// TIA Portal V17 export
// export: Created 2022-05-07T16:38:47.6768571Z, ExportSetting WithDefaults, DisplayName Totally Integrated Automation Portal, DisplayVersion V17 Update 3, DisplayName TIA Portal Openness, DisplayVersion V17 Update 3, DisplayName TIA Portal Version Control Interface, DisplayVersion V17, DisplayName TIA Portal Test Suite Advanced, DisplayVersion V17 Update 1, DisplayName SINAMICS Startdrive Advanced, DisplayVersion V17 Update2, DisplayName SINAMICS Startdrive G130, G150, S120, S150, SINAMICS MV, S210, DisplayVersion V17 Update2, DisplayName SINAMICS Startdrive G110M, G120, G120C, G120D, G120P, G115D, DisplayVersion V17 Update2, DisplayName STEP 7 Professional, DisplayVersion V17 Update 3, DisplayName STEP 7 Safety, DisplayVersion V17, DisplayName WinCC UA Professional, DisplayVersion V17 Update 3
FUNCTION_BLOCK "FB_ORG_ASSI"   // FB5, LAD
{ S7_Optimized_Access := 'TRUE' }
VERSION : 0.1
// stored: AutoNumber true, IsIECCheckEnabled false, IsRetainMemResEnabled false, MemoryReserve 100, SetENOAutomatically false, UDAEnableTagReadback false
   VAR
      CTRL_ASSE_STD_MA { S7_SetPoint := 'True'} : "CTRL_ASSE_STD";
      CTRL_ASSE_STD_MR { S7_SetPoint := 'True'} : "CTRL_ASSE_STD";
      CTRL_ASSE_STD_MS { S7_SetPoint := 'True'} : "CTRL_ASSE_STD";
      CTRL_ASSE_STD_ME { S7_SetPoint := 'True'} : "CTRL_ASSE_STD";
   END_VAR
BEGIN

REGION Network 1: RESET ALLARMI
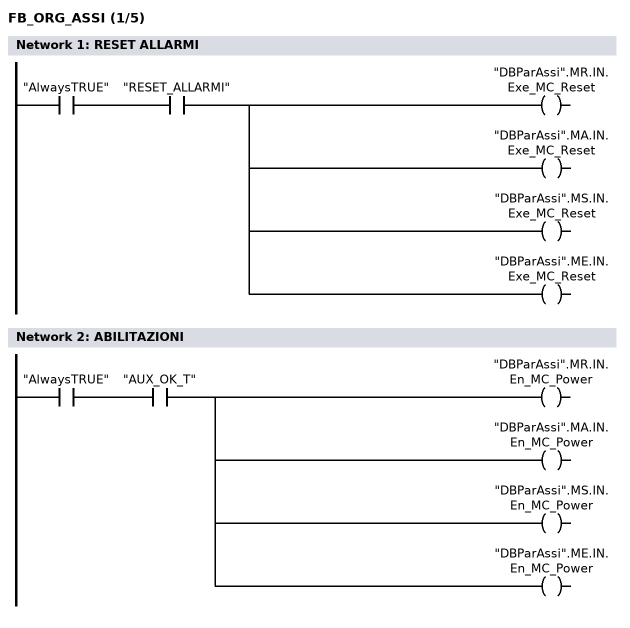
   RUNG wire#powerrail
      Contact( "AlwaysTRUE" )
      Contact( "RESET_ALLARMI" )
      wire#w1
      Coil( "DBParAssi".MR.IN.Exe_MC_Reset )
   END_RUNG
   RUNG wire#w1
      Coil( "DBParAssi".MA.IN.Exe_MC_Reset )
   END_RUNG
   RUNG wire#w1
      Coil( "DBParAssi".MS.IN.Exe_MC_Reset )
   END_RUNG
   RUNG wire#w1
      Coil( "DBParAssi".ME.IN.Exe_MC_Reset )
   END_RUNG
   // the same network as SCL:
   "DBParAssi".MR.IN.Exe_MC_Reset := "AlwaysTRUE" AND "RESET_ALLARMI";
   "DBParAssi".MA.IN.Exe_MC_Reset := "DBParAssi".MR.IN.Exe_MC_Reset;
   "DBParAssi".MS.IN.Exe_MC_Reset := "DBParAssi".MR.IN.Exe_MC_Reset;
   "DBParAssi".ME.IN.Exe_MC_Reset := "DBParAssi".MR.IN.Exe_MC_Reset;
END_REGION

REGION Network 2: ABILITAZIONI
   RUNG wire#powerrail
      Contact( "AlwaysTRUE" )
      Contact( "AUX_OK_T" )
      wire#w1
      Coil( "DBParAssi".MR.IN.En_MC_Power )
   END_RUNG
   RUNG wire#w1
      Coil( "DBParAssi".MA.IN.En_MC_Power )
   END_RUNG
   RUNG wire#w1
      Coil( "DBParAssi".MS.IN.En_MC_Power )
   END_RUNG
   RUNG wire#w1
      Coil( "DBParAssi".ME.IN.En_MC_Power )
   END_RUNG
   // the same network as SCL:
   "DBParAssi".MR.IN.En_MC_Power := "AlwaysTRUE" AND "AUX_OK_T";
   "DBParAssi".MA.IN.En_MC_Power := "DBParAssi".MR.IN.En_MC_Power;
   "DBParAssi".MS.IN.En_MC_Power := "DBParAssi".MR.IN.En_MC_Power;
   "DBParAssi".ME.IN.En_MC_Power := "DBParAssi".MR.IN.En_MC_Power;
END_REGION

REGION Network 3: ISTANZA MR
   // homing attivo = 3
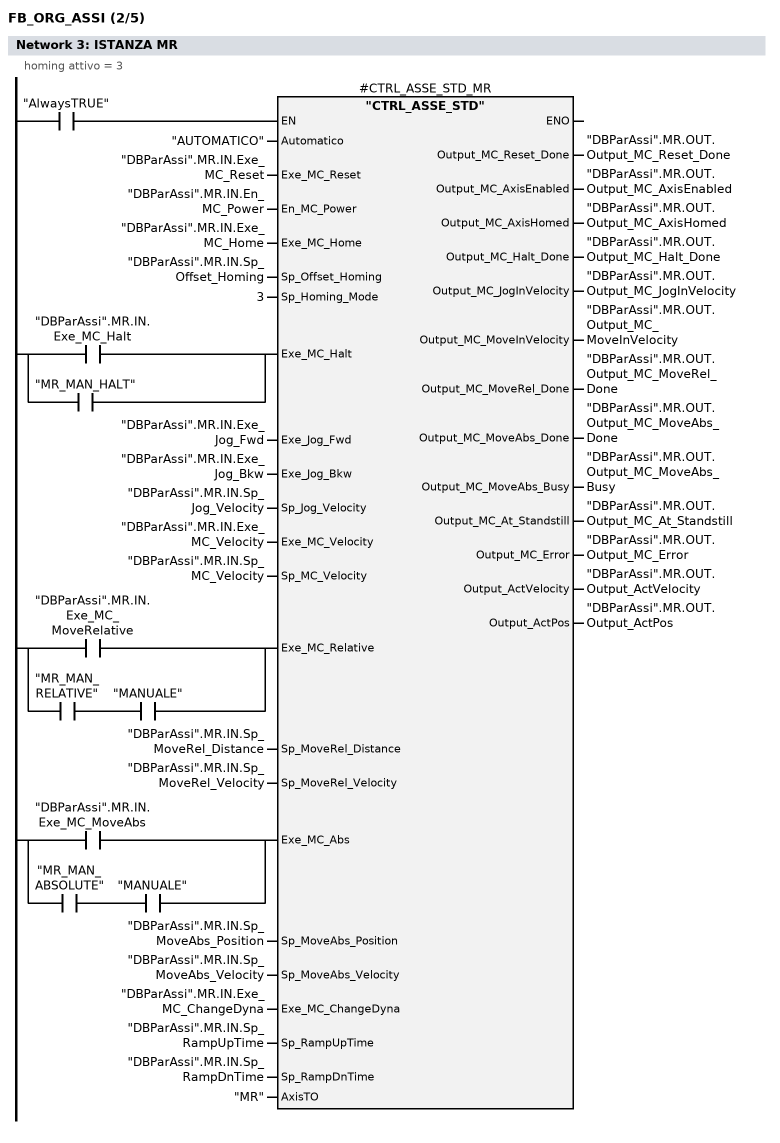
   RUNG wire#powerrail
      Contact( "AlwaysTRUE" )
      #CTRL_ASSE_STD_MR(Exe_MC_Halt := wire#w1, Exe_MC_Relative := wire#w2, Exe_MC_Abs := wire#w3, Automatico := "AUTOMATICO", Exe_MC_Reset := "DBParAssi".MR.IN.Exe_MC_Reset, En_MC_Power := "DBParAssi".MR.IN.En_MC_Power, Exe_MC_Home := "DBParAssi".MR.IN.Exe_MC_Home, Sp_Offset_Homing := "DBParAssi".MR.IN.Sp_Offset_Homing, Sp_Homing_Mode := 3, Exe_Jog_Fwd := "DBParAssi".MR.IN.Exe_Jog_Fwd, Exe_Jog_Bkw := "DBParAssi".MR.IN.Exe_Jog_Bkw, Sp_Jog_Velocity := "DBParAssi".MR.IN.Sp_Jog_Velocity, Exe_MC_Velocity := "DBParAssi".MR.IN.Exe_MC_Velocity, Sp_MC_Velocity := "DBParAssi".MR.IN.Sp_MC_Velocity, Sp_MoveRel_Distance := "DBParAssi".MR.IN.Sp_MoveRel_Distance, Sp_MoveRel_Velocity := "DBParAssi".MR.IN.Sp_MoveRel_Velocity, Sp_MoveAbs_Position := "DBParAssi".MR.IN.Sp_MoveAbs_Position, Sp_MoveAbs_Velocity := "DBParAssi".MR.IN.Sp_MoveAbs_Velocity, Exe_MC_ChangeDyna := "DBParAssi".MR.IN.Exe_MC_ChangeDyna, Sp_RampUpTime := "DBParAssi".MR.IN.Sp_RampUpTime, Sp_RampDnTime := "DBParAssi".MR.IN.Sp_RampDnTime, AxisTO := "MR", Output_MC_Reset_Done => "DBParAssi".MR.OUT.Output_MC_Reset_Done, Output_MC_AxisEnabled => "DBParAssi".MR.OUT.Output_MC_AxisEnabled, Output_MC_AxisHomed => "DBParAssi".MR.OUT.Output_MC_AxisHomed, Output_MC_Halt_Done => "DBParAssi".MR.OUT.Output_MC_Halt_Done, Output_MC_JogInVelocity => "DBParAssi".MR.OUT.Output_MC_JogInVelocity, Output_MC_MoveInVelocity => "DBParAssi".MR.OUT.Output_MC_MoveInVelocity, Output_MC_MoveRel_Done => "DBParAssi".MR.OUT.Output_MC_MoveRel_Done, Output_MC_MoveAbs_Done => "DBParAssi".MR.OUT.Output_MC_MoveAbs_Done, Output_MC_MoveAbs_Busy => "DBParAssi".MR.OUT.Output_MC_MoveAbs_Busy, Output_MC_At_Standstill => "DBParAssi".MR.OUT.Output_MC_At_Standstill, Output_MC_Error => "DBParAssi".MR.OUT.Output_MC_Error, Output_ActVelocity => "DBParAssi".MR.OUT.Output_ActVelocity, Output_ActPos => "DBParAssi".MR.OUT.Output_ActPos)
   END_RUNG
   RUNG wire#powerrail
      Contact( "DBParAssi".MR.IN.Exe_MC_Halt )
   END_RUNG wire#w1
   RUNG wire#powerrail
      Contact( "MR_MAN_HALT" )
   END_RUNG wire#w1
   RUNG wire#powerrail
      Contact( "DBParAssi".MR.IN.Exe_MC_MoveRelative )
   END_RUNG wire#w2
   RUNG wire#powerrail
      Contact( "MR_MAN_RELATIVE" )
      Contact( "MANUALE" )
   END_RUNG wire#w2
   RUNG wire#powerrail
      Contact( "DBParAssi".MR.IN.Exe_MC_MoveAbs )
   END_RUNG wire#w3
   RUNG wire#powerrail
      Contact( "MR_MAN_ABSOLUTE" )
      Contact( "MANUALE" )
   END_RUNG wire#w3
   // the same network as SCL:
   IF "AlwaysTRUE" THEN
       #CTRL_ASSE_STD_MR(Automatico := "AUTOMATICO",   // "CTRL_ASSE_STD"
                         Exe_MC_Reset := "DBParAssi".MR.IN.Exe_MC_Reset,
                         En_MC_Power := "DBParAssi".MR.IN.En_MC_Power,
                         Exe_MC_Home := "DBParAssi".MR.IN.Exe_MC_Home,
                         Sp_Offset_Homing := "DBParAssi".MR.IN.Sp_Offset_Homing,
                         Sp_Homing_Mode := 3,
                         Exe_MC_Halt := "DBParAssi".MR.IN.Exe_MC_Halt OR "MR_MAN_HALT",
                         Exe_Jog_Fwd := "DBParAssi".MR.IN.Exe_Jog_Fwd,
                         Exe_Jog_Bkw := "DBParAssi".MR.IN.Exe_Jog_Bkw,
                         Sp_Jog_Velocity := "DBParAssi".MR.IN.Sp_Jog_Velocity,
                         Exe_MC_Velocity := "DBParAssi".MR.IN.Exe_MC_Velocity,
                         Sp_MC_Velocity := "DBParAssi".MR.IN.Sp_MC_Velocity,
                         Exe_MC_Relative := "DBParAssi".MR.IN.Exe_MC_MoveRelative OR ("MR_MAN_RELATIVE" AND "MANUALE"),
                         Sp_MoveRel_Distance := "DBParAssi".MR.IN.Sp_MoveRel_Distance,
                         Sp_MoveRel_Velocity := "DBParAssi".MR.IN.Sp_MoveRel_Velocity,
                         Exe_MC_Abs := "DBParAssi".MR.IN.Exe_MC_MoveAbs OR ("MR_MAN_ABSOLUTE" AND "MANUALE"),
                         Sp_MoveAbs_Position := "DBParAssi".MR.IN.Sp_MoveAbs_Position,
                         Sp_MoveAbs_Velocity := "DBParAssi".MR.IN.Sp_MoveAbs_Velocity,
                         Exe_MC_ChangeDyna := "DBParAssi".MR.IN.Exe_MC_ChangeDyna,
                         Sp_RampUpTime := "DBParAssi".MR.IN.Sp_RampUpTime,
                         Sp_RampDnTime := "DBParAssi".MR.IN.Sp_RampDnTime,
                         AxisTO := "MR",
                         Output_MC_Reset_Done => "DBParAssi".MR.OUT.Output_MC_Reset_Done,
                         Output_MC_AxisEnabled => "DBParAssi".MR.OUT.Output_MC_AxisEnabled,
                         Output_MC_AxisHomed => "DBParAssi".MR.OUT.Output_MC_AxisHomed,
                         Output_MC_Halt_Done => "DBParAssi".MR.OUT.Output_MC_Halt_Done,
                         Output_MC_JogInVelocity => "DBParAssi".MR.OUT.Output_MC_JogInVelocity,
                         Output_MC_MoveInVelocity => "DBParAssi".MR.OUT.Output_MC_MoveInVelocity,
                         Output_MC_MoveRel_Done => "DBParAssi".MR.OUT.Output_MC_MoveRel_Done,
                         Output_MC_MoveAbs_Done => "DBParAssi".MR.OUT.Output_MC_MoveAbs_Done,
                         Output_MC_MoveAbs_Busy => "DBParAssi".MR.OUT.Output_MC_MoveAbs_Busy,
                         Output_MC_At_Standstill => "DBParAssi".MR.OUT.Output_MC_At_Standstill,
                         Output_MC_Error => "DBParAssi".MR.OUT.Output_MC_Error,
                         Output_ActVelocity => "DBParAssi".MR.OUT.Output_ActVelocity,
                         Output_ActPos => "DBParAssi".MR.OUT.Output_ActPos);
   END_IF;
END_REGION

REGION Network 4: ISTANZA MA
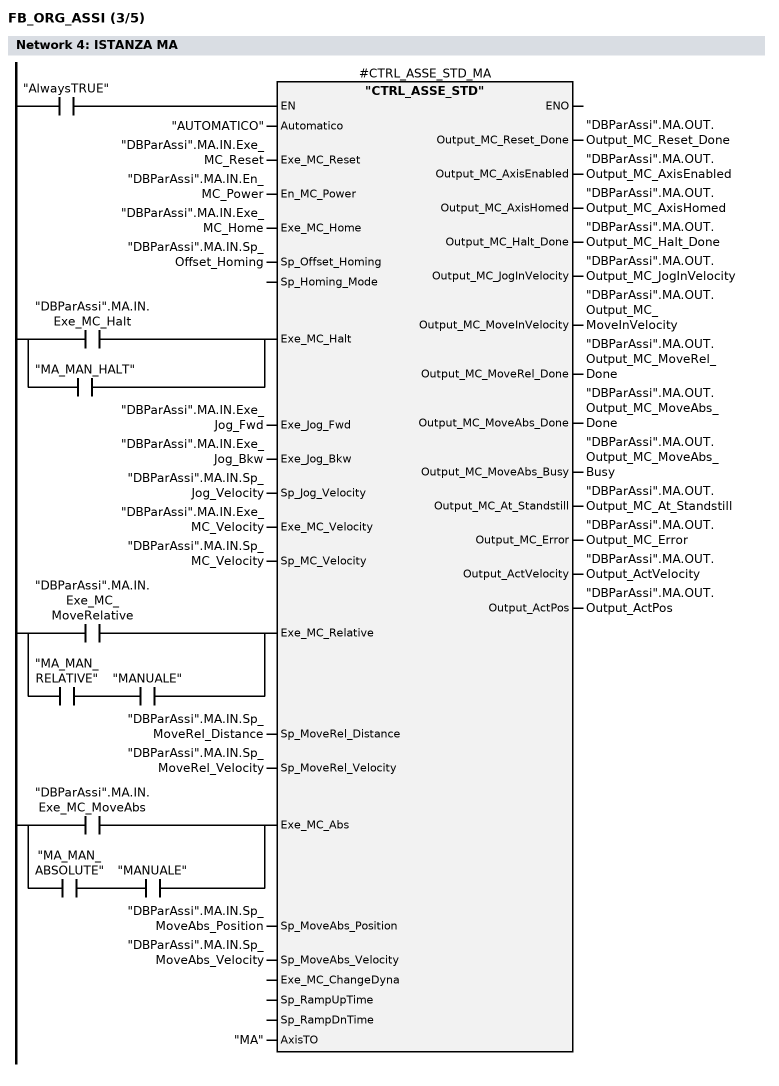
   RUNG wire#powerrail
      Contact( "AlwaysTRUE" )
      #CTRL_ASSE_STD_MA(Exe_MC_Halt := wire#w1, Exe_MC_Relative := wire#w2, Exe_MC_Abs := wire#w3, Automatico := "AUTOMATICO", Exe_MC_Reset := "DBParAssi".MA.IN.Exe_MC_Reset, En_MC_Power := "DBParAssi".MA.IN.En_MC_Power, Exe_MC_Home := "DBParAssi".MA.IN.Exe_MC_Home, Sp_Offset_Homing := "DBParAssi".MA.IN.Sp_Offset_Homing, Sp_Homing_Mode :=, Exe_Jog_Fwd := "DBParAssi".MA.IN.Exe_Jog_Fwd, Exe_Jog_Bkw := "DBParAssi".MA.IN.Exe_Jog_Bkw, Sp_Jog_Velocity := "DBParAssi".MA.IN.Sp_Jog_Velocity, Exe_MC_Velocity := "DBParAssi".MA.IN.Exe_MC_Velocity, Sp_MC_Velocity := "DBParAssi".MA.IN.Sp_MC_Velocity, Sp_MoveRel_Distance := "DBParAssi".MA.IN.Sp_MoveRel_Distance, Sp_MoveRel_Velocity := "DBParAssi".MA.IN.Sp_MoveRel_Velocity, Sp_MoveAbs_Position := "DBParAssi".MA.IN.Sp_MoveAbs_Position, Sp_MoveAbs_Velocity := "DBParAssi".MA.IN.Sp_MoveAbs_Velocity, Exe_MC_ChangeDyna :=, Sp_RampUpTime :=, Sp_RampDnTime :=, AxisTO := "MA", Output_MC_Reset_Done => "DBParAssi".MA.OUT.Output_MC_Reset_Done, Output_MC_AxisEnabled => "DBParAssi".MA.OUT.Output_MC_AxisEnabled, Output_MC_AxisHomed => "DBParAssi".MA.OUT.Output_MC_AxisHomed, Output_MC_Halt_Done => "DBParAssi".MA.OUT.Output_MC_Halt_Done, Output_MC_JogInVelocity => "DBParAssi".MA.OUT.Output_MC_JogInVelocity, Output_MC_MoveInVelocity => "DBParAssi".MA.OUT.Output_MC_MoveInVelocity, Output_MC_MoveRel_Done => "DBParAssi".MA.OUT.Output_MC_MoveRel_Done, Output_MC_MoveAbs_Done => "DBParAssi".MA.OUT.Output_MC_MoveAbs_Done, Output_MC_MoveAbs_Busy => "DBParAssi".MA.OUT.Output_MC_MoveAbs_Busy, Output_MC_At_Standstill => "DBParAssi".MA.OUT.Output_MC_At_Standstill, Output_MC_Error => "DBParAssi".MA.OUT.Output_MC_Error, Output_ActVelocity => "DBParAssi".MA.OUT.Output_ActVelocity, Output_ActPos => "DBParAssi".MA.OUT.Output_ActPos)
   END_RUNG
   RUNG wire#powerrail
      Contact( "DBParAssi".MA.IN.Exe_MC_Halt )
   END_RUNG wire#w1
   RUNG wire#powerrail
      Contact( "MA_MAN_HALT" )
   END_RUNG wire#w1
   RUNG wire#powerrail
      Contact( "DBParAssi".MA.IN.Exe_MC_MoveRelative )
   END_RUNG wire#w2
   RUNG wire#powerrail
      Contact( "MA_MAN_RELATIVE" )
      Contact( "MANUALE" )
   END_RUNG wire#w2
   RUNG wire#powerrail
      Contact( "DBParAssi".MA.IN.Exe_MC_MoveAbs )
   END_RUNG wire#w3
   RUNG wire#powerrail
      Contact( "MA_MAN_ABSOLUTE" )
      Contact( "MANUALE" )
   END_RUNG wire#w3
   // the same network as SCL:
   IF "AlwaysTRUE" THEN
       #CTRL_ASSE_STD_MA(Automatico := "AUTOMATICO",   // "CTRL_ASSE_STD"
                         Exe_MC_Reset := "DBParAssi".MA.IN.Exe_MC_Reset,
                         En_MC_Power := "DBParAssi".MA.IN.En_MC_Power,
                         Exe_MC_Home := "DBParAssi".MA.IN.Exe_MC_Home,
                         Sp_Offset_Homing := "DBParAssi".MA.IN.Sp_Offset_Homing,
                         Exe_MC_Halt := "DBParAssi".MA.IN.Exe_MC_Halt OR "MA_MAN_HALT",
                         Exe_Jog_Fwd := "DBParAssi".MA.IN.Exe_Jog_Fwd,
                         Exe_Jog_Bkw := "DBParAssi".MA.IN.Exe_Jog_Bkw,
                         Sp_Jog_Velocity := "DBParAssi".MA.IN.Sp_Jog_Velocity,
                         Exe_MC_Velocity := "DBParAssi".MA.IN.Exe_MC_Velocity,
                         Sp_MC_Velocity := "DBParAssi".MA.IN.Sp_MC_Velocity,
                         Exe_MC_Relative := "DBParAssi".MA.IN.Exe_MC_MoveRelative OR ("MA_MAN_RELATIVE" AND "MANUALE"),
                         Sp_MoveRel_Distance := "DBParAssi".MA.IN.Sp_MoveRel_Distance,
                         Sp_MoveRel_Velocity := "DBParAssi".MA.IN.Sp_MoveRel_Velocity,
                         Exe_MC_Abs := "DBParAssi".MA.IN.Exe_MC_MoveAbs OR ("MA_MAN_ABSOLUTE" AND "MANUALE"),
                         Sp_MoveAbs_Position := "DBParAssi".MA.IN.Sp_MoveAbs_Position,
                         Sp_MoveAbs_Velocity := "DBParAssi".MA.IN.Sp_MoveAbs_Velocity,
                         AxisTO := "MA",
                         Output_MC_Reset_Done => "DBParAssi".MA.OUT.Output_MC_Reset_Done,
                         Output_MC_AxisEnabled => "DBParAssi".MA.OUT.Output_MC_AxisEnabled,
                         Output_MC_AxisHomed => "DBParAssi".MA.OUT.Output_MC_AxisHomed,
                         Output_MC_Halt_Done => "DBParAssi".MA.OUT.Output_MC_Halt_Done,
                         Output_MC_JogInVelocity => "DBParAssi".MA.OUT.Output_MC_JogInVelocity,
                         Output_MC_MoveInVelocity => "DBParAssi".MA.OUT.Output_MC_MoveInVelocity,
                         Output_MC_MoveRel_Done => "DBParAssi".MA.OUT.Output_MC_MoveRel_Done,
                         Output_MC_MoveAbs_Done => "DBParAssi".MA.OUT.Output_MC_MoveAbs_Done,
                         Output_MC_MoveAbs_Busy => "DBParAssi".MA.OUT.Output_MC_MoveAbs_Busy,
                         Output_MC_At_Standstill => "DBParAssi".MA.OUT.Output_MC_At_Standstill,
                         Output_MC_Error => "DBParAssi".MA.OUT.Output_MC_Error,
                         Output_ActVelocity => "DBParAssi".MA.OUT.Output_ActVelocity,
                         Output_ActPos => "DBParAssi".MA.OUT.Output_ActPos);
   END_IF;
END_REGION

REGION Network 5 (SCL): ISTANZA MA SCL

   // #CTRL_ASSE_STD_MA(Exe_MC_Reset:="DBParAssi".MA.IN.Exe_MC_Reset,
   //                         En_MC_Power:="DBParAssi".MA.IN.En_MC_Power,
   //                         Exe_MC_Home:="DBParAssi".MA.IN.Exe_MC_Home,
   //                         Sp_Offset_Homing:="DBParAssi".MA.IN.Sp_Offset_Homing,
   //                         Exe_MC_Halt:="DBParAssi".MA.IN.Exe_MC_Halt,
   //                         Exe_Jog_Fwd:="DBParAssi".MA.IN.Exe_Jog_Fwd,
   //                         Exe_Jog_Bkw:="DBParAssi".MA.IN.Exe_Jog_Bkw,
   //                         Sp_Jog_Velocity:="DBParAssi".MA.IN.Sp_Jog_Velocity,
   //                         Exe_MC_Velocity:="DBParAssi".MA.IN.Exe_MC_Velocity,
   //                         Sp_MC_Velocity:="DBParAssi".MA.IN.Sp_MC_Velocity,
   //                         Exe_MC_Relative:="DBParAssi".MA.IN.Exe_MC_MoveRelative,
   //                         Sp_MoveRel_Distance:="DBParAssi".MA.IN.Sp_MoveRel_Distance,
   //                         Sp_MoveRel_Velocity:="DBParAssi".MA.IN.Sp_MoveRel_Velocity,
   //                         Exe_MC_Abs:="DBParAssi".MA.IN.Exe_MC_MoveAbs,
   //                         Sp_MoveAbs_Position:="DBParAssi".MA.IN.Sp_MoveAbs_Position,
   //                         Sp_MoveAbs_Velocity:="DBParAssi".MA.IN.Sp_MoveAbs_Velocity,
   //                         Output_MC_Reset_Done=>"DBParAssi".MA.OUT.Output_MC_Reset_Done,
   //                         Output_MC_AxisEnabled=>"DBParAssi".MA.OUT.Output_MC_AxisEnabled,
   //                         Output_MC_AxisHomed=>"DBParAssi".MA.OUT.Output_MC_AxisHomed,
   //                         Output_MC_Halt_Done=>"DBParAssi".MA.OUT.Output_MC_Halt_Done,
   //                         Output_MC_JogInVelocity=>"DBParAssi".MA.OUT.Output_MC_Reset_Done,
   //                         Output_MC_MoveInVelocity=>"DBParAssi".MA.OUT.Output_MC_MoveInVelocity,
   //                         Output_MC_MoveRel_Done=>"DBParAssi".MA.OUT.Output_MC_MoveRel_Done,
   //                         Output_MC_MoveAbs_Done=>"DBParAssi".MA.OUT.Output_MC_MoveAbs_Done,
   //                         Output_MC_MoveAbs_Busy=>"DBParAssi".MA.OUT.Output_MC_MoveAbs_Busy,
   //                         Output_MC_At_Standstill=>"DBParAssi".MA.OUT.Output_MC_Reset_Done,
   //                         Output_MC_Error=>"DBParAssi".MA.OUT.Output_MC_Error,
   //                         Output_ActVelocity=>"DBParAssi".MA.OUT.Output_ActVelocity,
   //                         Output_ActPos=>"DBParAssi".MA.OUT.Output_ActPos,
   //                         AxisTO:="MA");
END_REGION

REGION Network 6: ISTANZA MS
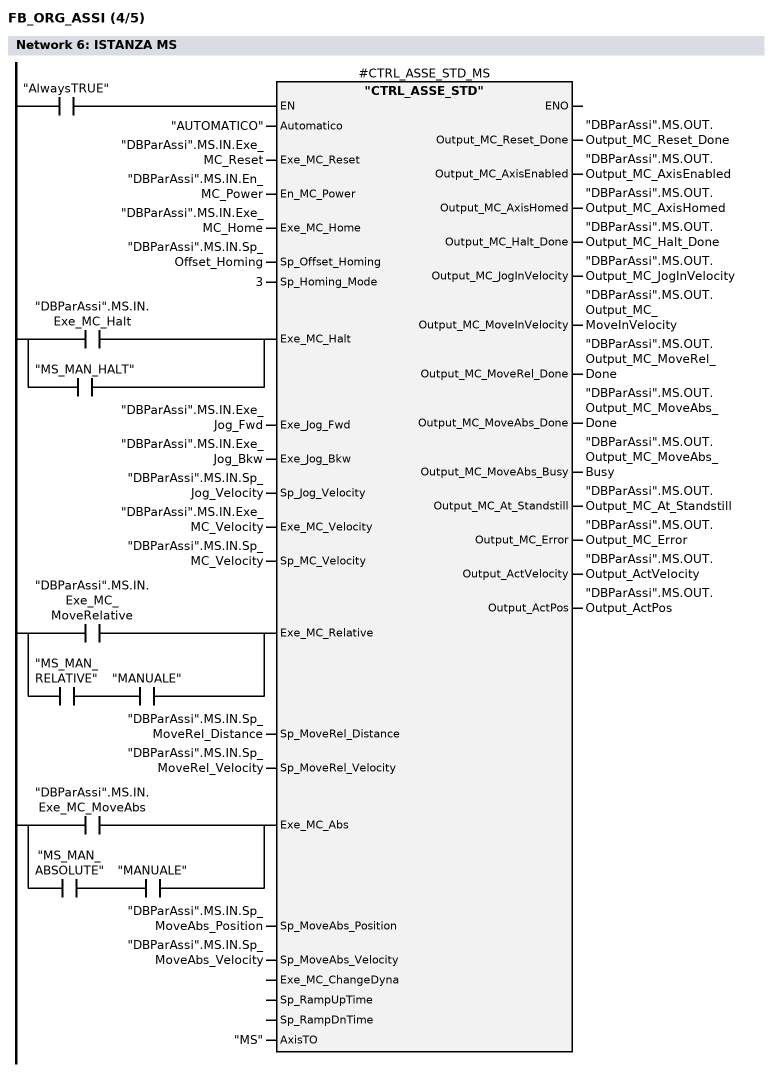
   RUNG wire#powerrail
      Contact( "AlwaysTRUE" )
      #CTRL_ASSE_STD_MS(Exe_MC_Halt := wire#w1, Exe_MC_Relative := wire#w2, Exe_MC_Abs := wire#w3, Automatico := "AUTOMATICO", Exe_MC_Reset := "DBParAssi".MS.IN.Exe_MC_Reset, En_MC_Power := "DBParAssi".MS.IN.En_MC_Power, Exe_MC_Home := "DBParAssi".MS.IN.Exe_MC_Home, Sp_Offset_Homing := "DBParAssi".MS.IN.Sp_Offset_Homing, Sp_Homing_Mode := 3, Exe_Jog_Fwd := "DBParAssi".MS.IN.Exe_Jog_Fwd, Exe_Jog_Bkw := "DBParAssi".MS.IN.Exe_Jog_Bkw, Sp_Jog_Velocity := "DBParAssi".MS.IN.Sp_Jog_Velocity, Exe_MC_Velocity := "DBParAssi".MS.IN.Exe_MC_Velocity, Sp_MC_Velocity := "DBParAssi".MS.IN.Sp_MC_Velocity, Sp_MoveRel_Distance := "DBParAssi".MS.IN.Sp_MoveRel_Distance, Sp_MoveRel_Velocity := "DBParAssi".MS.IN.Sp_MoveRel_Velocity, Sp_MoveAbs_Position := "DBParAssi".MS.IN.Sp_MoveAbs_Position, Sp_MoveAbs_Velocity := "DBParAssi".MS.IN.Sp_MoveAbs_Velocity, Exe_MC_ChangeDyna :=, Sp_RampUpTime :=, Sp_RampDnTime :=, AxisTO := "MS", Output_MC_Reset_Done => "DBParAssi".MS.OUT.Output_MC_Reset_Done, Output_MC_AxisEnabled => "DBParAssi".MS.OUT.Output_MC_AxisEnabled, Output_MC_AxisHomed => "DBParAssi".MS.OUT.Output_MC_AxisHomed, Output_MC_Halt_Done => "DBParAssi".MS.OUT.Output_MC_Halt_Done, Output_MC_JogInVelocity => "DBParAssi".MS.OUT.Output_MC_JogInVelocity, Output_MC_MoveInVelocity => "DBParAssi".MS.OUT.Output_MC_MoveInVelocity, Output_MC_MoveRel_Done => "DBParAssi".MS.OUT.Output_MC_MoveRel_Done, Output_MC_MoveAbs_Done => "DBParAssi".MS.OUT.Output_MC_MoveAbs_Done, Output_MC_MoveAbs_Busy => "DBParAssi".MS.OUT.Output_MC_MoveAbs_Busy, Output_MC_At_Standstill => "DBParAssi".MS.OUT.Output_MC_At_Standstill, Output_MC_Error => "DBParAssi".MS.OUT.Output_MC_Error, Output_ActVelocity => "DBParAssi".MS.OUT.Output_ActVelocity, Output_ActPos => "DBParAssi".MS.OUT.Output_ActPos)
   END_RUNG
   RUNG wire#powerrail
      Contact( "DBParAssi".MS.IN.Exe_MC_Halt )
   END_RUNG wire#w1
   RUNG wire#powerrail
      Contact( "MS_MAN_HALT" )
   END_RUNG wire#w1
   RUNG wire#powerrail
      Contact( "DBParAssi".MS.IN.Exe_MC_MoveRelative )
   END_RUNG wire#w2
   RUNG wire#powerrail
      Contact( "MS_MAN_RELATIVE" )
      Contact( "MANUALE" )
   END_RUNG wire#w2
   RUNG wire#powerrail
      Contact( "DBParAssi".MS.IN.Exe_MC_MoveAbs )
   END_RUNG wire#w3
   RUNG wire#powerrail
      Contact( "MS_MAN_ABSOLUTE" )
      Contact( "MANUALE" )
   END_RUNG wire#w3
   // the same network as SCL:
   IF "AlwaysTRUE" THEN
       #CTRL_ASSE_STD_MS(Automatico := "AUTOMATICO",   // "CTRL_ASSE_STD"
                         Exe_MC_Reset := "DBParAssi".MS.IN.Exe_MC_Reset,
                         En_MC_Power := "DBParAssi".MS.IN.En_MC_Power,
                         Exe_MC_Home := "DBParAssi".MS.IN.Exe_MC_Home,
                         Sp_Offset_Homing := "DBParAssi".MS.IN.Sp_Offset_Homing,
                         Sp_Homing_Mode := 3,
                         Exe_MC_Halt := "DBParAssi".MS.IN.Exe_MC_Halt OR "MS_MAN_HALT",
                         Exe_Jog_Fwd := "DBParAssi".MS.IN.Exe_Jog_Fwd,
                         Exe_Jog_Bkw := "DBParAssi".MS.IN.Exe_Jog_Bkw,
                         Sp_Jog_Velocity := "DBParAssi".MS.IN.Sp_Jog_Velocity,
                         Exe_MC_Velocity := "DBParAssi".MS.IN.Exe_MC_Velocity,
                         Sp_MC_Velocity := "DBParAssi".MS.IN.Sp_MC_Velocity,
                         Exe_MC_Relative := "DBParAssi".MS.IN.Exe_MC_MoveRelative OR ("MS_MAN_RELATIVE" AND "MANUALE"),
                         Sp_MoveRel_Distance := "DBParAssi".MS.IN.Sp_MoveRel_Distance,
                         Sp_MoveRel_Velocity := "DBParAssi".MS.IN.Sp_MoveRel_Velocity,
                         Exe_MC_Abs := "DBParAssi".MS.IN.Exe_MC_MoveAbs OR ("MS_MAN_ABSOLUTE" AND "MANUALE"),
                         Sp_MoveAbs_Position := "DBParAssi".MS.IN.Sp_MoveAbs_Position,
                         Sp_MoveAbs_Velocity := "DBParAssi".MS.IN.Sp_MoveAbs_Velocity,
                         AxisTO := "MS",
                         Output_MC_Reset_Done => "DBParAssi".MS.OUT.Output_MC_Reset_Done,
                         Output_MC_AxisEnabled => "DBParAssi".MS.OUT.Output_MC_AxisEnabled,
                         Output_MC_AxisHomed => "DBParAssi".MS.OUT.Output_MC_AxisHomed,
                         Output_MC_Halt_Done => "DBParAssi".MS.OUT.Output_MC_Halt_Done,
                         Output_MC_JogInVelocity => "DBParAssi".MS.OUT.Output_MC_JogInVelocity,
                         Output_MC_MoveInVelocity => "DBParAssi".MS.OUT.Output_MC_MoveInVelocity,
                         Output_MC_MoveRel_Done => "DBParAssi".MS.OUT.Output_MC_MoveRel_Done,
                         Output_MC_MoveAbs_Done => "DBParAssi".MS.OUT.Output_MC_MoveAbs_Done,
                         Output_MC_MoveAbs_Busy => "DBParAssi".MS.OUT.Output_MC_MoveAbs_Busy,
                         Output_MC_At_Standstill => "DBParAssi".MS.OUT.Output_MC_At_Standstill,
                         Output_MC_Error => "DBParAssi".MS.OUT.Output_MC_Error,
                         Output_ActVelocity => "DBParAssi".MS.OUT.Output_ActVelocity,
                         Output_ActPos => "DBParAssi".MS.OUT.Output_ActPos);
   END_IF;
END_REGION

REGION Network 7: ISTANZA ME
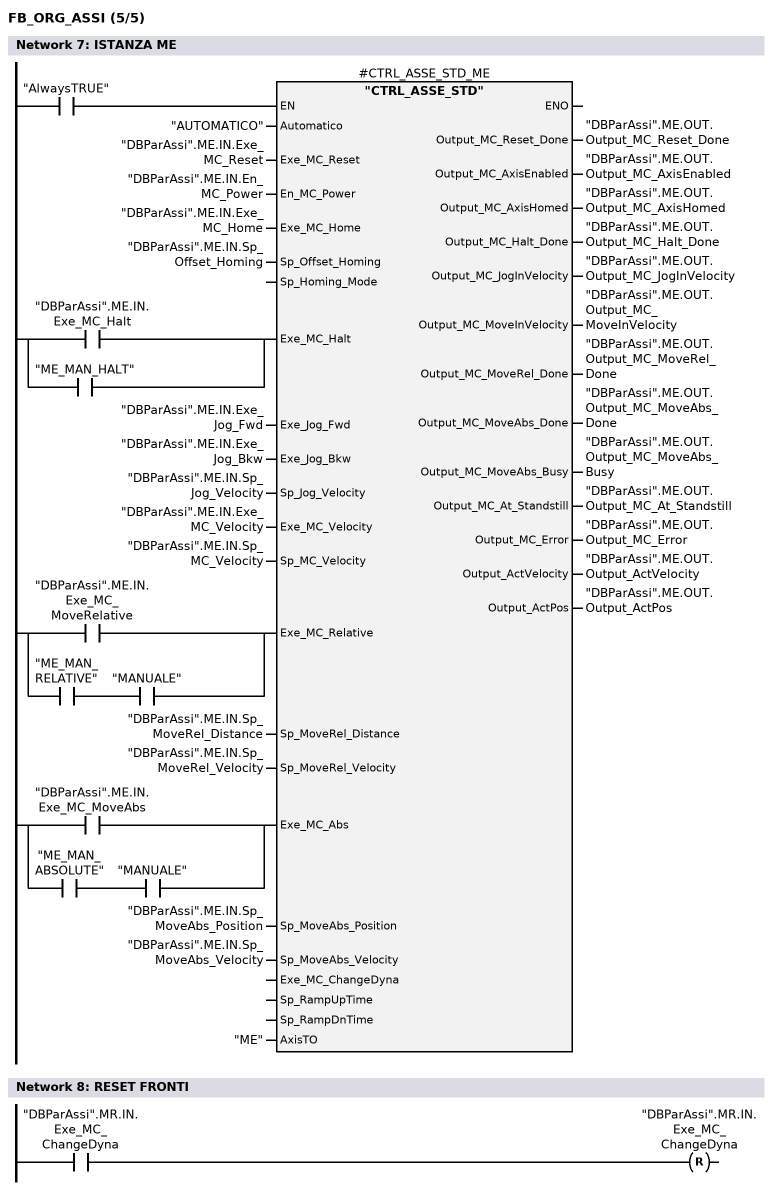
   RUNG wire#powerrail
      Contact( "AlwaysTRUE" )
      #CTRL_ASSE_STD_ME(Exe_MC_Halt := wire#w1, Exe_MC_Relative := wire#w2, Exe_MC_Abs := wire#w3, Automatico := "AUTOMATICO", Exe_MC_Reset := "DBParAssi".ME.IN.Exe_MC_Reset, En_MC_Power := "DBParAssi".ME.IN.En_MC_Power, Exe_MC_Home := "DBParAssi".ME.IN.Exe_MC_Home, Sp_Offset_Homing := "DBParAssi".ME.IN.Sp_Offset_Homing, Sp_Homing_Mode :=, Exe_Jog_Fwd := "DBParAssi".ME.IN.Exe_Jog_Fwd, Exe_Jog_Bkw := "DBParAssi".ME.IN.Exe_Jog_Bkw, Sp_Jog_Velocity := "DBParAssi".ME.IN.Sp_Jog_Velocity, Exe_MC_Velocity := "DBParAssi".ME.IN.Exe_MC_Velocity, Sp_MC_Velocity := "DBParAssi".ME.IN.Sp_MC_Velocity, Sp_MoveRel_Distance := "DBParAssi".ME.IN.Sp_MoveRel_Distance, Sp_MoveRel_Velocity := "DBParAssi".ME.IN.Sp_MoveRel_Velocity, Sp_MoveAbs_Position := "DBParAssi".ME.IN.Sp_MoveAbs_Position, Sp_MoveAbs_Velocity := "DBParAssi".ME.IN.Sp_MoveAbs_Velocity, Exe_MC_ChangeDyna :=, Sp_RampUpTime :=, Sp_RampDnTime :=, AxisTO := "ME", Output_MC_Reset_Done => "DBParAssi".ME.OUT.Output_MC_Reset_Done, Output_MC_AxisEnabled => "DBParAssi".ME.OUT.Output_MC_AxisEnabled, Output_MC_AxisHomed => "DBParAssi".ME.OUT.Output_MC_AxisHomed, Output_MC_Halt_Done => "DBParAssi".ME.OUT.Output_MC_Halt_Done, Output_MC_JogInVelocity => "DBParAssi".ME.OUT.Output_MC_JogInVelocity, Output_MC_MoveInVelocity => "DBParAssi".ME.OUT.Output_MC_MoveInVelocity, Output_MC_MoveRel_Done => "DBParAssi".ME.OUT.Output_MC_MoveRel_Done, Output_MC_MoveAbs_Done => "DBParAssi".ME.OUT.Output_MC_MoveAbs_Done, Output_MC_MoveAbs_Busy => "DBParAssi".ME.OUT.Output_MC_MoveAbs_Busy, Output_MC_At_Standstill => "DBParAssi".ME.OUT.Output_MC_At_Standstill, Output_MC_Error => "DBParAssi".ME.OUT.Output_MC_Error, Output_ActVelocity => "DBParAssi".ME.OUT.Output_ActVelocity, Output_ActPos => "DBParAssi".ME.OUT.Output_ActPos)
   END_RUNG
   RUNG wire#powerrail
      Contact( "DBParAssi".ME.IN.Exe_MC_Halt )
   END_RUNG wire#w1
   RUNG wire#powerrail
      Contact( "ME_MAN_HALT" )
   END_RUNG wire#w1
   RUNG wire#powerrail
      Contact( "DBParAssi".ME.IN.Exe_MC_MoveRelative )
   END_RUNG wire#w2
   RUNG wire#powerrail
      Contact( "ME_MAN_RELATIVE" )
      Contact( "MANUALE" )
   END_RUNG wire#w2
   RUNG wire#powerrail
      Contact( "DBParAssi".ME.IN.Exe_MC_MoveAbs )
   END_RUNG wire#w3
   RUNG wire#powerrail
      Contact( "ME_MAN_ABSOLUTE" )
      Contact( "MANUALE" )
   END_RUNG wire#w3
   // the same network as SCL:
   IF "AlwaysTRUE" THEN
       #CTRL_ASSE_STD_ME(Automatico := "AUTOMATICO",   // "CTRL_ASSE_STD"
                         Exe_MC_Reset := "DBParAssi".ME.IN.Exe_MC_Reset,
                         En_MC_Power := "DBParAssi".ME.IN.En_MC_Power,
                         Exe_MC_Home := "DBParAssi".ME.IN.Exe_MC_Home,
                         Sp_Offset_Homing := "DBParAssi".ME.IN.Sp_Offset_Homing,
                         Exe_MC_Halt := "DBParAssi".ME.IN.Exe_MC_Halt OR "ME_MAN_HALT",
                         Exe_Jog_Fwd := "DBParAssi".ME.IN.Exe_Jog_Fwd,
                         Exe_Jog_Bkw := "DBParAssi".ME.IN.Exe_Jog_Bkw,
                         Sp_Jog_Velocity := "DBParAssi".ME.IN.Sp_Jog_Velocity,
                         Exe_MC_Velocity := "DBParAssi".ME.IN.Exe_MC_Velocity,
                         Sp_MC_Velocity := "DBParAssi".ME.IN.Sp_MC_Velocity,
                         Exe_MC_Relative := "DBParAssi".ME.IN.Exe_MC_MoveRelative OR ("ME_MAN_RELATIVE" AND "MANUALE"),
                         Sp_MoveRel_Distance := "DBParAssi".ME.IN.Sp_MoveRel_Distance,
                         Sp_MoveRel_Velocity := "DBParAssi".ME.IN.Sp_MoveRel_Velocity,
                         Exe_MC_Abs := "DBParAssi".ME.IN.Exe_MC_MoveAbs OR ("ME_MAN_ABSOLUTE" AND "MANUALE"),
                         Sp_MoveAbs_Position := "DBParAssi".ME.IN.Sp_MoveAbs_Position,
                         Sp_MoveAbs_Velocity := "DBParAssi".ME.IN.Sp_MoveAbs_Velocity,
                         AxisTO := "ME",
                         Output_MC_Reset_Done => "DBParAssi".ME.OUT.Output_MC_Reset_Done,
                         Output_MC_AxisEnabled => "DBParAssi".ME.OUT.Output_MC_AxisEnabled,
                         Output_MC_AxisHomed => "DBParAssi".ME.OUT.Output_MC_AxisHomed,
                         Output_MC_Halt_Done => "DBParAssi".ME.OUT.Output_MC_Halt_Done,
                         Output_MC_JogInVelocity => "DBParAssi".ME.OUT.Output_MC_JogInVelocity,
                         Output_MC_MoveInVelocity => "DBParAssi".ME.OUT.Output_MC_MoveInVelocity,
                         Output_MC_MoveRel_Done => "DBParAssi".ME.OUT.Output_MC_MoveRel_Done,
                         Output_MC_MoveAbs_Done => "DBParAssi".ME.OUT.Output_MC_MoveAbs_Done,
                         Output_MC_MoveAbs_Busy => "DBParAssi".ME.OUT.Output_MC_MoveAbs_Busy,
                         Output_MC_At_Standstill => "DBParAssi".ME.OUT.Output_MC_At_Standstill,
                         Output_MC_Error => "DBParAssi".ME.OUT.Output_MC_Error,
                         Output_ActVelocity => "DBParAssi".ME.OUT.Output_ActVelocity,
                         Output_ActPos => "DBParAssi".ME.OUT.Output_ActPos);
   END_IF;
END_REGION

REGION Network 8: RESET FRONTI
   RUNG wire#powerrail
      Contact( "DBParAssi".MR.IN.Exe_MC_ChangeDyna )
      R_Coil( "DBParAssi".MR.IN.Exe_MC_ChangeDyna )
   END_RUNG
   // the same network as SCL:
   IF "DBParAssi".MR.IN.Exe_MC_ChangeDyna THEN "DBParAssi".MR.IN.Exe_MC_ChangeDyna := FALSE; END_IF;
END_REGION
END_FUNCTION_BLOCK
